RoboDK station: Blank workstation not merged.rdk

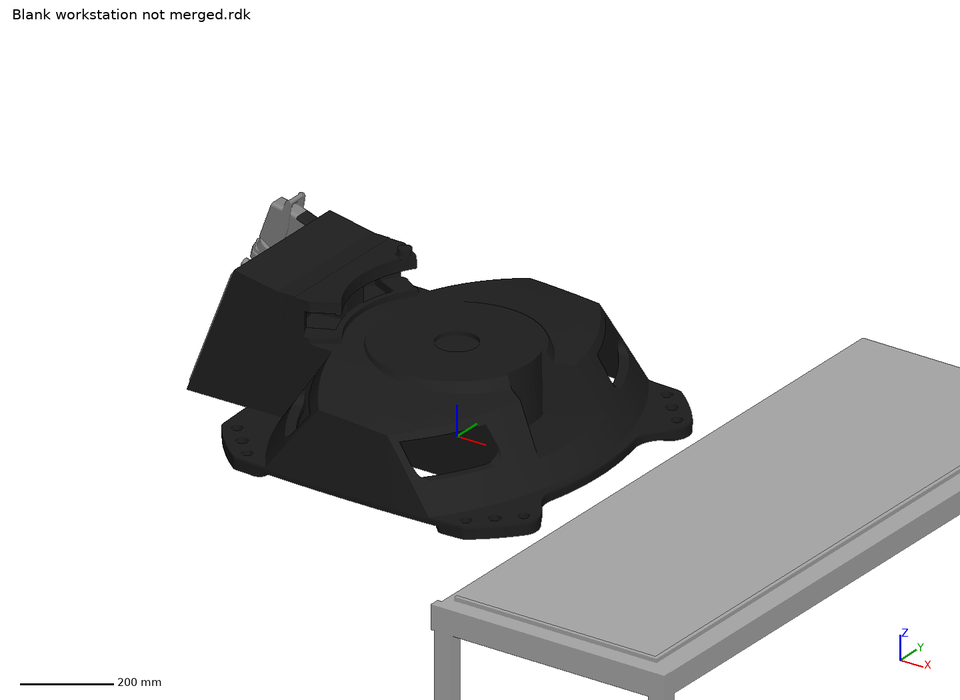
[picture v0: the station drawn from its stored meshes, robots at their saved joint values, targets as dots, program paths as lines]
Station Blank workstation not merged (saved by RoboDK 5.2.3). Poses are relative to the parent item; angles as X-Y-Z fixed-axis rotations.
  - frame KUKA KR 210 R2700 extra Base at (0, 0, 0) mm
    - robot KUKA KR 210 R2700 extra: 6 axes, payload 210 kg, reach 2696 mm, repeatability 0.06 mm, weight 1068 kg
        joint limits [-185, -140, -120, -350, -125, -350] to [185, -5, 155, 350, 125, 350]; home [0, -90, 90, 0, 0, 0]; saved at [102.054, -9.211, 11.208, -275.332, 1.867, -91.819]
  - object FrameLeg at (520, -780, -400) mm, size 40 x 40 x 400 mm, geometry from FrameLeg.stl
  - object FramePLate at (800, 45, 0) mm, size 600 x 1600 x 25 mm, geometry from FramePLate.stl
  - object FrameTop at (800, 0, 0) mm, size 610 x 1605 x 60 mm, geometry from FrameTop.stl
  - object FrameLeg at (1080, -780, -400) mm, size 40 x 40 x 400 mm, geometry from FrameLeg.stl
  - object FrameLeg at (1080, 780, -400) mm, size 40 x 40 x 400 mm, geometry from FrameLeg.stl
  - object FrameLeg at (520, 780, -400) mm, size 40 x 40 x 400 mm, geometry from FrameLeg.stl
